// Mitsubishi GX Works2 project: 230928-001-SET E RESET   PLC: Q03UDV

// task Task_01 (event TRUE, interval 0, priority 31): POU_01

PROGRAM POU_01
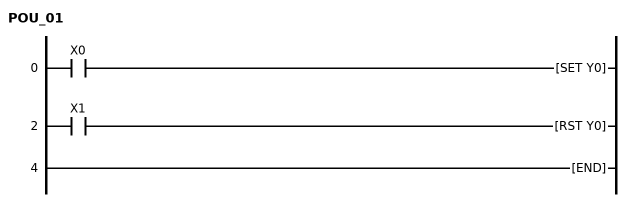
0     LD      X0
      SET     Y0
2     LD      X1
      RST     Y0
4     END
END_PROGRAM
